FUNCTION_BLOCK FB_loading
VAR_INPUT
	pre_tote_status			: ToteStatus;//roller -1 totestatus=ready
	next_tote_status		: ToteStatus;//roller +1 totestatus=empty
	bRun					: BOOL;
	bReset					: BOOL;
	bSafety					: BOOL;
END_VAR
VAR_OUTPUT
	ready_recive		: BOOL;
	tote_recivied_current		: BOOL;//current roller recived the tote
END_VAR
VAR
	current_tote_status	: ToteStatus;
	ton_timeout			: TON;	
	eStates				: E_LoadingStates := E_LoadingStates.IDLE;
	eStateTemp			: E_LoadingStates := E_LoadingStates.IDLE;
	iStateTemp			: INT;
	sStateTemp			: STRING;
	errorMessage		: STRING;
	xError				: BOOL;
	event				: ST_EVENT;
	rt_error			: R_TRIG;
///////////////hardware define//////////////////	
	roller_x					: Roller_x;
	roller_y					: Roller_y;
	photo_sensor_tote_detection	: BOOL;
	EDM_KA7						: BOOL;
	mcAxis	 					: FB_MotionAxis_MC;
	st_mcAxis					: ST_MotionAxis_MC;
	AxisRef						: AXIS_REF;	
END_VAR
VAR CONSTANT
	rPos_load	: REAL := 0;
	rPos_unload	: REAL := 1;
	sComponent_name			: STRING := 'fb_loading';
END_VAR

M_mapping();


rt_error(CLK:=(roller_x.roller.err OR roller_y.roller.err OR st_mcAxis.mcReadStatus.Error) 
	AND MAIN.eState<>E_SystemManager.RESET_SAFETY);//roller will trig error while power on
IF rt_error.Q THEN
	xError	:= TRUE;
	eStates	:= E_LoadingStates.ERROR;
END_IF

METHOD M_agingTest : BOOL
VAR_INPUT
	
END_VAR
M_AgingTest	:= FALSE;
//////////////////////////////////////////////////////////timeout//////////////////////////////////////////
iStateTemp	:= eStateTemp;
ton_timeout();
IF eStates<>E_LoadingStates.IDLE AND eStates<>E_LoadingStates.ERROR THEN
	IF eStateTemp=eStates THEN
		ton_timeout.IN	:=TRUE;
	ELSE
		ton_timeout.IN	:=FALSE;
		eStateTemp	:= eStates;
	END_IF
ELSE
	ton_timeout.IN	:=FALSE;
END_IF
IF ton_timeout.Q THEN	
	ton_timeout.IN	:=FALSE;
	CASE eStates OF
		E_LoadingStates.AGING_STATE_0:		
			errorMessage	:= CONCAT('wait loading timeout.->fb_loading ',INT_TO_STRING(iStateTemp));
		E_LoadingStates.AGING_STATE_1:		
			errorMessage	:= CONCAT('wait unloading timeout.->fb_loading ',INT_TO_STRING(iStateTemp));
	END_CASE
	IF eStates<>E_LoadingStates.WAIT AND eStates<>E_LoadingStates.WAIT_1 THEN
		eStates	:= E_LoadingStates.ERROR;
	END_IF
END_IF
CASE eStates OF
	E_LoadingStates.IDLE:
		eStates	:= E_LoadingStates.AGING_STATE_0;
	E_LoadingStates.AGING_STATE_0:
		ton_timeout.PT	:= T#10S;
		roller_x.roller.forward		:= TRUE;
		roller_y.roller.forward		:= TRUE;
		roller_y.roller.backward	:= FALSE;		
		st_mcAxis.mcMoveAbsolute.Execute	:= TRUE;						
		st_mcAxis.rActualPosSet	:= 800;
		st_mcAxis.rVelocitySet	:= 200;
		IF st_mcAxis.mcMoveAbsolute.Done THEN
			eStates	:= E_LoadingStates.WAIT;
		END_IF			
	E_LoadingStates.WAIT:
		roller_x.roller.forward		:= FALSE;
		roller_x.roller.backward	:= FALSE;
		roller_y.roller.forward		:= FALSE;
		roller_y.roller.backward	:= FALSE;	
		st_mcAxis.mcMoveAbsolute.Execute	:= FALSE;
		ton_timeout.PT	:= T#2S;
		IF ton_timeout.Q THEN
			eStates	:= E_LoadingStates.AGING_STATE_1;
		END_IF
	E_LoadingStates.AGING_STATE_1:
		ton_timeout.PT	:= T#10S;
		roller_x.roller.backward	:= TRUE;
		roller_y.roller.forward		:= TRUE;
		roller_y.roller.backward	:= TRUE;			
		st_mcAxis.mcMoveAbsolute.Execute	:= TRUE;						
		st_mcAxis.rActualPosSet	:= 0;
		st_mcAxis.rVelocitySet	:= 200;
		IF st_mcAxis.mcMoveAbsolute.Done THEN
			eStates	:= E_LoadingStates.WAIT_1;
		END_IF	
	E_LoadingStates.WAIT_1:
		roller_x.roller.forward		:= FALSE;
		roller_x.roller.backward	:= FALSE;
		roller_y.roller.forward		:= FALSE;
		roller_y.roller.backward	:= FALSE;	
		st_mcAxis.mcMoveAbsolute.Execute	:= FALSE;	
		ton_timeout.PT	:= T#2S;
		IF ton_timeout.Q THEN
			eStates	:= E_LoadingStates.IDLE;
		END_IF		
	E_LoadingStates.DONE:
		;
	E_LoadingStates.ERROR:
		;
	
END_CASE
END_METHOD

METHOD M_init : BOOL
VAR_INPUT
END_VAR
VAR
END_VAR
M_init	:= FALSE;
xError	:= FALSE;
eStates	:=E_LoadingStates.IDLE;
M_init	:= TRUE;
END_METHOD

METHOD M_load : BOOL
VAR_INPUT
END_VAR
END_METHOD

METHOD M_mapping : BOOL
VAR_INPUT
END_VAR
event.sTime	:= MAIN.Temp_str;
event.sComponent_name	:= sComponent_name;
/////////////////////////////////////digital input////////////////////////////////////////
roller_x.photo_sensor_mute_left			:= G_IO.arDI[3].Ch[0];
roller_x.roller.err						:= G_IO.arDI[3].Ch[1];
roller_x.photo_sensor_mute_right		:= G_IO.arDI[3].Ch[2];
roller_y.roller.err						:= G_IO.arDI[3].Ch[3];
roller_y.photo_sensor[0]				:= G_IO.arDI[3].Ch[4];
roller_y.photo_sensor[1]				:= G_IO.arDI[3].Ch[5];
photo_sensor_tote_detection				:= G_IO.arDI[3].Ch[6];
EDM_KA7									:= G_IO.arDI[3].Ch[7];

/////////////////////////////////////digital output////////////////////////////////////////
G_IO.arDO[3].Ch[0]	:= roller_x.roller.forward;
G_IO.arDO[3].Ch[1]	:= roller_x.roller.backward;
G_IO.arDO[3].Ch[2]	:= roller_y.roller.forward;
G_IO.arDO[3].Ch[3]	:= roller_y.roller.backward;




/////////////////////////////////////axis config////////////////////////////////////////
mcAxis
(
	ZSN		:=  TRUE OR st_mcAxis.xHoming, //TODO link to digital input
	ZSP		:=  TRUE OR st_mcAxis.xHoming, //TODO link to digital input
	IN_OUT	:= st_mcAxis	, 
	AXIS	:= AxisRef	, 
);
st_mcAxis.bPosSensorShow	:= TRUE;
st_mcAxis.bNegSensorShow	:= TRUE;
st_mcAxis.rMaxAcceleration	:= 50000;
st_mcAxis.rMaxDeceleration	:= 50000;
st_mcAxis.rMaxJerk			:= 500000;
st_mcAxis.rAcceleration	:= 2500;
st_mcAxis.rDeceleration	:= 2500;
st_mcAxis.rJerk			:= 12500;
st_mcAxis.rMaxVelocity		:= 100;
st_mcAxis.rMaxDistance		:= 50;
st_mcAxis.bPosSen	:= TRUE ;//TODO link to digital input
st_mcAxis.bNegSen	:= TRUE ;//TODO link to digital input
st_mcAxis.mcHome.bCalibrationCam	:= TRUE;//TODO link to digital input origin
st_mcAxis.bPositionSensor	:= TRUE;//TODO link to digital input origin
st_mcAxis.bdirFW	:= TRUE;
st_mcAxis.sNetID := '192.168.11.159.5.1';
st_mcAxis.nSlaveAddr	:= 1017;


//
IF MAIN.firstCycle THEN
	st_mcAxis.mcPower.Enable	:= TRUE;
END_IF
END_METHOD

METHOD M_reset : BOOL
VAR_INPUT
END_VAR
M_reset	:= FALSE;
ton_timeout.IN	:= FALSE;
st_mcAxis.mcStop.Execute	:= FALSE;
st_mcAxis.mcReset.Execute	:= TRUE;
IF xError THEN
	IF eStates<>E_LoadingStates.IDLE THEN
		eStates	:= eStateTemp;//continue
	END_IF
	xError	:= FALSE;
ELSE
	M_reset	:= TRUE;
END_IF
END_METHOD

METHOD M_run : BOOL
VAR_INPUT
END_VAR
M_run	:= FALSE;
event.sMethod	:= 'M_run';
//////////////////////////////////////////////////////////current_tote status//////////////////////////////////////////
IF photo_sensor_tote_detection AND NOT(roller_x.photo_sensor_mute_left OR roller_x.photo_sensor_mute_right) THEN
	current_tote_status	:= ToteStatus.READY;
END_IF
IF NOT(roller_x.photo_sensor_mute_left OR roller_x.photo_sensor_mute_right 
	OR roller_y.photo_sensor[0] OR roller_y.photo_sensor[1]OR roller_y.roller.sensor) THEN
	current_tote_status	:= ToteStatus.EMPTY;
END_IF
//////////////////////////////////////////////////////////timeout//////////////////////////////////////////
IF 	eStates=E_LoadingStates.LIFT_POSITION_UNLOAD
	OR eStates=	E_LoadingStates.ROLLER_UNLOAD		
	OR eStates=	E_LoadingStates.WAIT_RIGHT_MUTE_OFF THEN
	IF MAIN.application.tote_subsystem.cmd<>OrderToteCommand.LOAD THEN//not count timer and run until cmd=load
		RETURN;
	END_IF
END_IF
		
		
iStateTemp	:= eStateTemp;
sStateTemp	:= INT_TO_STRING(iStateTemp);
ton_timeout();
IF eStates<>E_LoadingStates.IDLE AND eStates<>E_LoadingStates.ERROR THEN
	IF eStateTemp=eStates THEN
		ton_timeout.IN	:=TRUE;
	ELSE
		ton_timeout.IN	:=FALSE;
		IF GVL.bAck_stop THEN
			roller_x.roller.forward	:= FALSE;
			RETURN;		
		END_IF
		eStateTemp	:= eStates;
	END_IF
ELSE
	ton_timeout.IN	:=FALSE;
END_IF
IF ton_timeout.Q THEN	
	ton_timeout.IN	:=FALSE;
	CASE eStates OF		
		E_LoadingStates.LOADING:	
			event.sEventType	:= 'error';
			event.sEvent_MSG	:=  CONCAT('LOADING ','timeout');
			event.sStepID		:= sStateTemp;
		E_LoadingStates.LIFT_POSITION_LOAD:		
			event.sEventType	:= 'error';
			event.sEvent_MSG	:=  CONCAT('LIFT_POSITION_LOAD ','timeout');
			event.sStepID		:= sStateTemp;
		E_LoadingStates.ROLLER_LOAD:
			event.sEventType	:= 'error';
			event.sEvent_MSG	:=  CONCAT('ROLLER_LOAD ','timeout');
			event.sStepID		:= sStateTemp;
		E_LoadingStates.WAIT_LEFT_MUTE_OFF:
			event.sEventType	:= 'error';
			event.sEvent_MSG	:=  CONCAT('WAIT_LEFT_MUTE_OFF ','timeout');
			event.sStepID		:= sStateTemp;
		E_LoadingStates.UNLOADING:	
			event.sEventType	:= 'error';
			event.sEvent_MSG	:=  CONCAT('UNLOADING ','timeout');
			event.sStepID		:= sStateTemp;
		E_LoadingStates.LIFT_POSITION_UNLOAD:	
				event.sEventType	:= 'error';
			event.sEvent_MSG	:=  CONCAT('sStateTemp ','timeout');
			event.sStepID		:= sStateTemp;
		E_LoadingStates.ROLLER_UNLOAD:
			event.sEventType	:= 'error';
			event.sEvent_MSG	:=  CONCAT('ROLLER_UNLOAD ','timeout');
			event.sStepID		:= sStateTemp;	
		E_LoadingStates.WAIT_RIGHT_MUTE_OFF:
			event.sEventType	:= 'error';
			event.sEvent_MSG	:=  CONCAT('WAIT_RIGHT_MUTE_OFF ','timeout');
			event.sStepID		:= sStateTemp;	
	END_CASE
	IF eStates<>E_LoadingStates.WAIT AND eStates<>E_LoadingStates.DETECTION THEN
		eStates	:= E_LoadingStates.ERROR;
		Event_add(event);
	END_IF
END_IF

CASE eStates OF 
		E_LoadingStates.IDLE:	
			eStates	:= E_LoadingStates.INIT;
		E_LoadingStates.INIT:
			eStates	:= E_LoadingStates.WAIT;
		E_LoadingStates.WAIT:
			eStates	:= E_LoadingStates.DETECTION;
		E_LoadingStates.DETECTION:
			st_mcAxis.mcMoveAbsolute.Execute	:= FALSE;
			roller_x.roller.forward	:= FALSE;
			ton_timeout.PT	:= T#10S;
			IF pre_tote_status=ToteStatus.READY AND current_tote_status=ToteStatus.EMPTY THEN
				eStates	:= E_LoadingStates.LOADING;
			END_IF
			IF next_tote_status=ToteStatus.EMPTY AND current_tote_status=ToteStatus.READY AND MAIN.application.tote_subsystem.cmd=OrderToteCommand.LOAD THEN
				eStates	:= E_LoadingStates.UNLOADING;
			END_IF				
		E_LoadingStates.LOADING:	
			eStates	:= E_LoadingStates.LIFT_POSITION_LOAD;
		E_LoadingStates.LIFT_POSITION_LOAD:				
			st_mcAxis.mcMoveAbsolute.Execute	:= TRUE;						
			st_mcAxis.rActualPosSet	:= rPos_load;
			st_mcAxis.rVelocitySet	:= 20;
			IF st_mcAxis.mcMoveAbsolute.Done THEN
				st_mcAxis.mcMoveAbsolute.Execute	:= FALSE;
				eStates	:= E_LoadingStates.ROLLER_LOAD;
			END_IF	
		E_LoadingStates.ROLLER_LOAD:
			roller_x.roller.forward	:= TRUE;
			IF photo_sensor_tote_detection THEN
				eStates	:= E_LoadingStates.WAIT_LEFT_MUTE_OFF;
			END_IF
		E_LoadingStates.WAIT_LEFT_MUTE_OFF:
			roller_x.roller.forward	:= TRUE;
			IF NOT roller_x.photo_sensor_mute_left THEN
				roller_x.roller.forward	:= FALSE;
				eStates	:= E_LoadingStates.DETECTION;
			END_IF	
		E_LoadingStates.UNLOADING:	
			eStates	:= E_LoadingStates.LIFT_POSITION_UNLOAD;
		E_LoadingStates.LIFT_POSITION_UNLOAD:
			st_mcAxis.mcMoveAbsolute.Execute	:= TRUE;						
			st_mcAxis.rActualPosSet	:= rPos_unload;
			st_mcAxis.rVelocitySet	:= 20;
			IF st_mcAxis.mcMoveAbsolute.Done THEN
				st_mcAxis.mcMoveAbsolute.Execute	:= FALSE;
				eStates	:= E_LoadingStates.ROLLER_UNLOAD;
			END_IF	
		E_LoadingStates.ROLLER_UNLOAD:
			roller_x.roller.forward	:= TRUE;
			IF NOT photo_sensor_tote_detection THEN
				eStates	:= E_LoadingStates.WAIT_RIGHT_MUTE_OFF;
			END_IF			
		E_LoadingStates.WAIT_RIGHT_MUTE_OFF:
			roller_x.roller.forward	:= TRUE;
			IF NOT roller_x.photo_sensor_mute_right THEN
				roller_x.roller.forward	:= FALSE;
				eStates	:= E_LoadingStates.DETECTION;
			END_IF				
		E_LoadingStates.DONE:			
			eStates	:= E_LoadingStates.IDLE;
		E_LoadingStates.ERROR:
			st_mcAxis.mcMoveAbsolute.Execute	:= FALSE;
			roller_x.roller.forward	:= FALSE;			
			xError	:=	TRUE;	
END_CASE
END_METHOD

METHOD M_runStart : BOOL
VAR_INPUT
END_VAR
M_runStart	:= FALSE;
st_mcAxis.mcPower.Enable	:= TRUE;
IF st_mcAxis.mcReadStatus.StandStill THEN
	M_runStart	:= TRUE;
END_IF
M_runStart	:= TRUE;
END_METHOD

METHOD M_safetyEvent : BOOL
VAR_INPUT
END_VAR
M_safetyEvent	:= FALSE;

roller_x.roller.forward		:= FALSE;
roller_x.roller.backward	:= FALSE;
roller_y.roller.forward		:= FALSE;
roller_y.roller.backward	:= FALSE;
st_mcAxis.mcMoveAbsolute.Execute	:= FALSE;
st_mcAxis.mcStop.Execute	:= TRUE;

M_safetyEvent	:= TRUE;
END_METHOD

METHOD M_unload : BOOL
VAR_INPUT
END_VAR
END_METHOD

END_FUNCTION_BLOCK

(* stored: Version 1.1.0.1, ProductVersion 3.1.4024.12
   POU FB_loading: Id {e407b83c-c16b-4915-840f-648913a3d5a1}, SpecialFunc None
   Method M_agingTest: Id {75165e62-765c-445b-bb52-8f7e914ddba8}
   Method M_init: Id {8333a8c5-63e7-4729-acc2-82dfb9a83857}
   Method M_load: Id {381f8622-a963-4bbf-99cb-da0723814a76}
   Method M_mapping: Id {22e87662-5706-4a10-aeb7-20d6a2c5a8a9}
   Method M_reset: Id {da9a24c2-cd48-4508-98e7-e9ad8d66aac6}
   Method M_run: Id {05ac0d68-304e-43d6-8c1c-c552e8e88d14}
   Method M_runStart: Id {83ce8a34-c979-4038-95d4-da4d50b5c36e}
   Method M_safetyEvent: Id {1b31e517-8d93-44b8-81eb-24eec7bb0098}
   Method M_unload: Id {b4982e2c-1d77-4024-ae62-ea58585970e7} *)
